PROGRAM peddal
VAR
	//autonoom
	Autonoom : BOOL;
	SetAutonoom : BOOL;	
	
	//voor inleen pedal en rem
	RemIngedrukt : BOOL;
	InputNum AT%I* : INT;
	PercentagePedal : REAL;

	//Voor Motion
	fbReadXaxisStatus: MC_ReadStatus;
	triggerAutonoom: F_TRIG;
	LowMode : BOOL;
END_VAR

   triggerAutonoom(CLK:= SetAutonoom, Q=> );
Autonoom S= TriggerAutonoom.Q;
IF Autonoom THEN
	PercentagePedal := Scaling(Input:= InputNum, Imin:= 0, Imax:= 32767, Qmin:= 0, Qmax:= 100);
  Autonoom R= RemIngedrukt OR PercentagePedal > 10;
END_IF

IF LowMode THEN // als lowmode aan is, is maximum throtthe 50%
		IF PercentagePedal > 50 THEN
			PercentagePedal := 50;
		END_IF
END_IF

END_PROGRAM

(* stored: Version 1.1.0.1, ProductVersion 3.1.4024.3
   POU peddal: Id {8d2bd18b-9383-4735-8d16-06e116df72cb}, SpecialFunc None *)
